// TIA Portal project "ModbusTCPSever" (V14)

(* hardware
DEVICE "S7-1200 station_1"  S7-1200 Station
   slot 0: "Rack_0"  S7-1200 Rack  Rack  V1.0
   slot 1: "PLC_1"  CPU 1212C DC/DC/DC  6ES7 212-1AE40-0XB0  V4.2
*)

// ===== PLC "PLC_1"  CPU 1212C DC/DC/DC =====

VAR_GLOBAL   // PLC tag table "默认变量表"
   "mb_disconnect" AT %M10.0 : Bool;
   "mb_ndr" AT %M10.1 : Bool;
   "mb_dr" AT %M10.2 : Bool;
   "mb_error" AT %M10.3 : Bool;
   "mb_status" AT %MW12 : Word;
   "mb_en" AT %M10.4 : Bool;
   "Tag_1" AT %Q0.0 : Bool;
   "Tag_2" AT %Q0.2 : Bool;
   "Tag_3" AT %Q0.4 : Bool;
   "Tag_4" AT %Q0.6 : Bool;
END_VAR

DATA_BLOCK "HoldRegs"   // DB2
{ S7_Optimized_Access := 'FALSE' }
VERSION : 0.1
   VAR
      Data : Array[0..9] of Word;
   END_VAR
BEGIN
   Data[0] := 2021;
   Data[1] := 06;
   Data[2] := 04;
   Data[3] := 10;
   Data[4] := 33;
   Data[5] := 12;
END_DATA_BLOCK

DATA_BLOCK "ModbusSeverConfig"   // DB3
{ S7_Optimized_Access := 'TRUE' }
VERSION : 0.1
   VAR
      config : TCON_IP_v4;
   END_VAR
BEGIN
   config.InterfaceId := 64;
   config.ID := 1;
   config.RemoteAddress.ADDR[1] := 192;
   config.RemoteAddress.ADDR[2] := 168;
   config.RemoteAddress.ADDR[3] := 1;
   config.RemoteAddress.ADDR[4] := 1;
   config.RemotePort := 0;
   config.LocalPort := 502;
END_DATA_BLOCK

ORGANIZATION_BLOCK "Main"   // OB1, LAD, ProgramCycle
TITLE = "Main Program Sweep (Cycle)"
{ S7_Optimized_Access := 'TRUE' }
VERSION : 0.1
   VAR_INPUT
      Initial_Call : Bool;   // Initial call of this OB
      Remanence : Bool;   // =True, if remanent data are available
   END_VAR
   VAR_TEMP
      DisConnect : Bool;   // 0:被动连接；1:终止连接且status=0003
      WriteNewData : Bool;   // 0:无数据；1:有从新数据
      ReadNewData : Bool;   // 1：有读取新数据
      Error : Bool;   // 为1时出错
      Status : Word;   // 状态信息
   END_VAR
BEGIN

REGION Network 1
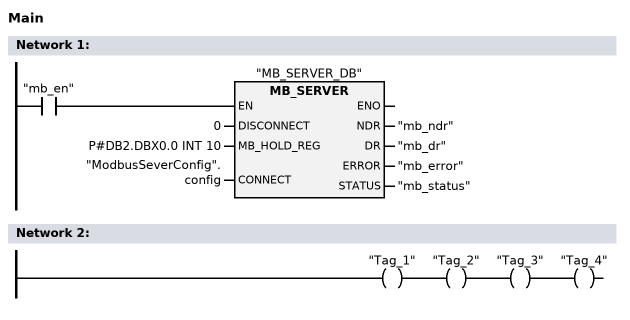
   IF "mb_en" THEN
       "MB_SERVER_DB"(DISCONNECT := 0,   // MB_SERVER
                      MB_HOLD_REG := P#DB2.DBX0.0 INT 10,
                      CONNECT := "ModbusSeverConfig".config,
                      NDR => "mb_ndr",
                      DR => "mb_dr",
                      ERROR => "mb_error",
                      STATUS => "mb_status");
   END_IF;
END_REGION

REGION Network 2
   RUNG wire#powerrail
      Coil( "Tag_1" )
      Coil( "Tag_2" )
      Coil( "Tag_3" )
      Coil( "Tag_4" )
   END_RUNG
   // the same network as SCL:
   "Tag_1" := TRUE;
   "Tag_2" := TRUE;
   "Tag_3" := TRUE;
   "Tag_4" := TRUE;
END_REGION
END_ORGANIZATION_BLOCK